Universal Robots PolyScope program: Short_PHomeToInvA.urp

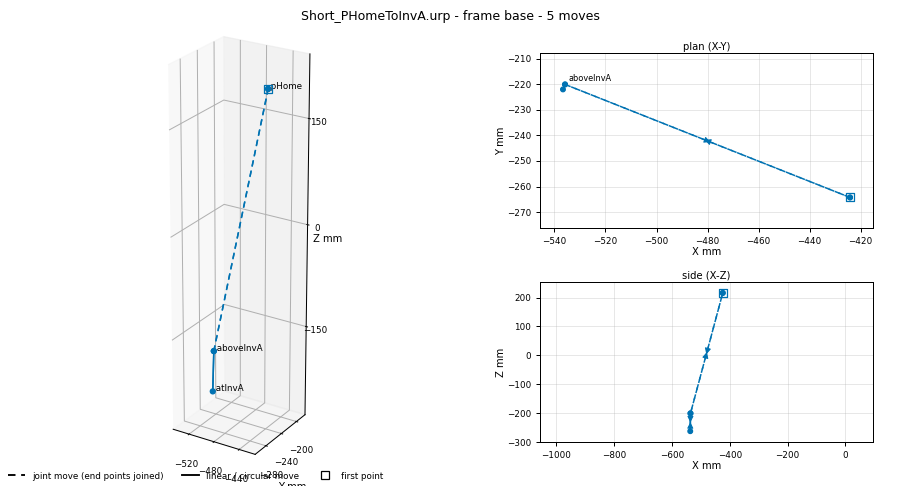
[picture p0: tool path of Short_PHomeToInvA.urp in frame base, 5 of 5 moves have a stored position in this frame; points joined in program order, loops and branches not executed]
Program Short_PHomeToInvA (installation=admin directory=/programs/THU_530PM/Final createdIn=3.8.0.61336 lastSavedIn=3.15.8.106339 robotSerialNumber=2015350925)
Calibrated DH parameters: a=[0, -0.425, -0.39225, 0, 0, 0]; d=[0.089159, 0, 0, 0.10915, 0.09465, 0.0823]; alpha=[1.570796, 0, 0, 1.570796, -1.570796, 0]; deltaTheta=[0, 0, 0, 0, 0, 0]
Robot Program (runOnlyOnce=true)
  Set DigitalOutput pin=digital_out[0]; digitalValue=1
  Wait Sleep waitTime=1
  Call _adminLinearIndex1
  Wait Sleep waitTime=1
  MoveJ speed 180 deg/s, acceleration 100 deg/s^2 (useActiveTCP=true)
    Waypoint pHome: TCP in base x=-424.177 y=-264.287 z=215.871 mm, rx=-1.1973 ry=-2.8917 rz=-0.0084 rad; joints [224.995, -90.007, -90.004, -90.013, 89.257, -0.019] deg; flange x=-422.26 y=-266.331 z=431.752 mm, rx=-1.1973 ry=-2.8917 rz=-0.0084 rad
    Waypoint aboveInvA: TCP in base x=-535.843 y=-220.007 z=-200.771 mm, rx=2.9366 ry=1.065 rz=-0.0096 rad; joints [212.702, -127.597, -109.536, -32.299, 90.919, 82.838] deg; flange x=-535.911 y=-215.937 z=15.091 mm, rx=2.9366 ry=1.065 rz=-0.0096 rad
  MoveL speed 250 mm/s, acceleration 500 mm/s^2 (useActiveTCP=true) feature=Base
    Waypoint atInvA: TCP in base x=-536.653 y=-221.96 z=-262.509 mm, rx=2.9366 ry=1.0649 rz=-0.0096 rad; joints [212.824, -135.386, -108.746, -25.298, 90.917, 82.963] deg; flange x=-536.721 y=-217.894 z=-46.647 mm, rx=2.9366 ry=1.0649 rz=-0.0096 rad
    Set DigitalOutput pin=digital_out[0]; digitalValue=0
    Wait Sleep waitTime=1
    Waypoint aboveInvA: motionParameters(blendRadius=0.01); TCP in base x=-535.843 y=-220.007 z=-200.771 mm, rx=2.9366 ry=1.065 rz=-0.0096 rad; joints [212.702, -127.597, -109.536, -32.299, 90.919, 82.838] deg; flange x=-535.911 y=-215.937 z=15.091 mm, rx=2.9366 ry=1.065 rz=-0.0096 rad
  MoveJ speed 180 deg/s, acceleration 100 deg/s^2 (useActiveTCP=true)
    Waypoint pHome: TCP in base x=-424.177 y=-264.287 z=215.871 mm, rx=-1.1973 ry=-2.8917 rz=-0.0084 rad; joints [224.995, -90.007, -90.004, -90.013, 89.257, -0.019] deg; flange x=-422.26 y=-266.331 z=431.752 mm, rx=-1.1973 ry=-2.8917 rz=-0.0084 rad
SubProgram -> _adminLinearIndex1
SubProgram _adminLinearIndex1 (keepSynchronizedWithDisk=false) programFile=/programs/me345_admin/_adminLinearIndex1.urp
  Folder Move_linear_slide_Index1
    var_1 := False
    Loop While (checkContinuously=false) expression=var_1≟ False
      var_1 := socket_open("10.241.34.48",4001)
    var_3 := 1
    Send := "s r0x24 21"
    Script: socket_send_string(Send)
    Script: socket_send_byte(13)
    Send_Reply := socket_read_string()
    Send := "s r0xca 0"
    Script: socket_send_string(Send)
    Script: socket_send_byte(13)
    Send_Reply := socket_read_string()
    Send := "t 1"
    Script: socket_send_string(Send)
    Script: socket_send_byte(13)
    Send_Reply := socket_read_string()
    Loop While (checkContinuously=false) expression=var_3≠0
      Send := "g r0xA0"
      Script: socket_send_string(Send)
      Script: socket_send_byte(13)
      var_3 := socket_get_var("v")
      Wait Sleep waitTime=0.1
    Script: socket_close()
    Script: sync()
